(* IEC 61131-3 sources: POMIRTS_lab3/AS/Library/LoopCont/V3.03.2, 3 files *)

(* ---- LoopCont.typ ---- *)
(********************************************************************
 * COPYRIGHT (C) BERNECKER + RAINER, AUSTRIA, A-5142 EGGELSBERG
 ********************************************************************
 * Library: LoopCont
 * File: LoopCont.typ
 * Created: 11.11.2003
 ********************************************************************
 * Global data types of library LoopCont
 ********************************************************************)

TYPE
	lcslimpid_par_typ : 	STRUCT
		Y_max : INT;
		Y_min : INT;
		Kp : REAL;
		Tn : REAL;
		Tv : REAL;
		Kfbk : REAL;
	END_STRUCT;
	lcpid_tune_addpar_typ : 	STRUCT
		t_max_tune : UDINT;
		dY_max : REAL;
		Tf_Tv : REAL;
		Kw : REAL;
		Kfbk : REAL;
		fbk_mode : USINT;
		d_mode : USINT;
		calc_mode : USINT;
	END_STRUCT;
	lcpid_tune_osc_options_typ : 	STRUCT
		osc_minAmplitude : INT;
		Q_min : REAL;
	END_STRUCT;
	lcpid_osc_val_typ : 	STRUCT
		X : INT;
		t : UDINT;
	END_STRUCT;
	lcpid_osc_per_typ : 	STRUCT
		max : lcpid_osc_val_typ;
		min : lcpid_osc_val_typ;
	END_STRUCT;
	lcpid_tune_osc_typ : 	STRUCT
		options : lcpid_tune_osc_options_typ;
		oscPhase : UINT;
		dir : SINT;
		Y_hi : INT;
		Y_lo : INT;
		i_maxPeriod : UINT;
		i_period : UINT;
		X_ampl : DINT;
		X_avg : DINT;
		X_min_avg : DINT;
		X_max_avg : DINT;
		Y_avg : DINT;
		deltaY : DINT;
		t_Ylohi : ARRAY[0..4] OF UDINT;
		t_Yhilo : ARRAY[0..4] OF UDINT;
		Q_act : REAL;
		a_wx : INT;
		amplitudeRatio : REAL;
		Ku : REAL;
		tPeriod : UDINT;
		period : ARRAY[0..4] OF lcpid_osc_per_typ;
	END_STRUCT;
	lcpid_tune_step_options_typ : 	STRUCT
		eqDeltaX : INT;
		eqDeltaWX : INT;
		eqDeltat : UDINT;
		evalDeltaX : INT;
		evalNfilter : UINT;
		exitNotMaxdXCount : UINT;
		exitdXRatio : UINT;
	END_STRUCT;
	lcpid_tune_step_typ : 	STRUCT
		options : lcpid_tune_step_options_typ;
		Y0 : INT;
		Y1 : INT;
		t_jump : UDINT;
		W : INT;
		X0 : INT;
		Xmax : INT;
		Xmin : INT;
		Xfiltered : DINT;
		deltaXok : BOOL;
		deltaWXok : BOOL;
		eqTime : UDINT;
		dir : SINT;
		deltaX : INT;
		X1 : INT;
		t1 : UDINT;
		t1set : BOOL;
		dX_dt : REAL;
		dX_dt_max : REAL;
		XmaxGrad : INT;
		maxX1 : INT;
		maxX2 : INT;
		maxt1 : UDINT;
		maxt2 : UDINT;
		tmaxGrad : UDINT;
		gainFactor : REAL;
		deadTime : UDINT;
		riseTime : UDINT;
		notMaxCount : UINT;
		gradientRatio : UINT;
		cycleTime : UDINT;
	END_STRUCT;
	lcdblpid_tune_typ : 	STRUCT
		P1_manualAdjust : INT;
		I1_manualAdjust : INT;
		D1_manualAdjust : INT;
		P2_manualAdjust : INT;
		I2_manualAdjust : INT;
		D2_manualAdjust : INT;
		X_min : INT;
		X_max : INT;
		X0 : INT;
		de_min : INT;
		Y0 : INT;
		Y1step : INT;
		Y2step : INT;
		tuneY1_opt : UDINT;
		tuneY2_opt : UDINT;
		tune_first : USINT;
		hyst : INT;
		measDelta : INT;
		osc_opt : lcpid_tune_osc_options_typ;
		step_opt : lcpid_tune_step_options_typ;
	END_STRUCT;
	lcdblpid_par_typ : 	STRUCT
		Y_max : INT;
		Y_min : INT;
		K_fact : INT;
		Kp : REAL;
		Tn : REAL;
		Tv : REAL;
	END_STRUCT;
	lcCurveByPoints_TabEntry_type : 	STRUCT
		x : INT;
		y : INT;
	END_STRUCT;
	lcpid_addPar_typ : 	STRUCT
		y_autotune_on : INT;
		y_autotune_off : INT;
		t_autotune_max : UDINT;
		diff_dx_max : INT;
		diff_dt_max : UDINT;
		osc_nrPeriods : UINT;
		osc_minAmplitude : INT;
		optSwitches : UINT;
		dY_max : REAL;
		Tf_Tv : REAL;
		Kw : REAL;
		Kfbk : REAL;
		fbk_mode : USINT;
		d_mode : USINT;
		calc_mode : USINT;
	END_STRUCT;
	lcpid_internal_typ : 	STRUCT
		size : UINT;
		valid : BOOL;
		autotune_addpar : lcpid_addPar_typ;
		Y_max : INT;
		Y_min : INT;
		dY_max1 : DINT;
		Kp1 : DINT;
		Kp_Tn_1 : DINT;
		Tv_Tf_1 : DINT;
		Tf_reciproc_1 : DINT;
		Kw1 : DINT;
		Kfbk_Kp_1 : DINT;
		fbk_mode : USINT;
		d_mode : USINT;
		calc_mode : USINT;
		prescalerPow2 : UINT;
		force_outmode : USINT;
		Y_force : INT;
		W : INT;
		X : INT;
		pid_init : USINT;
		dt : UDINT;
		Yp1 : DINT;
		Yp2 : DINT;
		dYi1 : DINT;
		dYi2 : DINT;
		Yi1 : DINT;
		Yi2 : DINT;
		dt_Tf_1 : DINT;
		a11 : DINT;
		a12 : DINT;
		a21 : DINT;
		a22 : DINT;
		Yd1 : DINT;
		Yd2 : DINT;
		Ytotal1 : DINT;
		Ytotal2 : DINT;
		Ylim1 : DINT;
		Ylim2 : DINT;
		Y1 : DINT;
		Y2 : DINT;
		e_fbk : DINT;
	END_STRUCT;
	lcpid_osc_typ : 	STRUCT
		i_maxPeriod : UINT;
		i_period : UINT;
		X_amplitude : DINT;
		amplitudeRatio : REAL;
		tPeriod : UDINT;
		period : ARRAY[0..4] OF lcpid_osc_per_typ;
	END_STRUCT;
	lcpid_procPar_typ : 	STRUCT
		size : UINT;
		valid : BOOL;
		stepResp_valid : BOOL;
		stepResp_v : REAL;
		stepResp_t_u : UDINT;
		stepResp_t_g : UDINT;
		osc_valid : BOOL;
		osc_amplitudeRatio : REAL;
		osc_tPeriod : UDINT;
		force_params : BOOL;
		Kp : REAL;
		Kp_tune : REAL;
		Tn : REAL;
		Tn_tune : REAL;
		Tv : REAL;
		Tv_tune : REAL;
	END_STRUCT;
	lcpid_old_typ : 	STRUCT
		processPar : lcpid_procPar_typ;
		P_manualAdjust : INT;
		I_manualAdjust : INT;
		D_manualAdjust : INT;
		Y_min : INT;
		Y_max : INT;
		dY_max : REAL;
		Tf_Tv : REAL;
		Kw : REAL;
		Kfbk : REAL;
		request : UDINT;
		time : UDINT;
		W : INT;
		fbk_mode : USINT;
		d_mode : USINT;
		enable : BOOL;
	END_STRUCT;
	lcpid_stepResp_typ : 	STRUCT
		W_old : INT;
		dW : INT;
		x_prev : INT;
		x_inflectionPt : INT;
		t_inflectionPt : UDINT;
		v : REAL;
		v_max : REAL;
		t_u : UDINT;
		x_pre : INT;
		x_max : INT;
	END_STRUCT;
	lcpid_diff_typ : 	STRUCT
		init : BOOL;
		x_old : INT;
		dx : INT;
		dt : UDINT;
		dx_dt : REAL;
	END_STRUCT;
END_TYPE

(* ---- LoopCont.fun ---- *)
(********************************************************************
 * COPYRIGHT (C) BERNECKER + RAINER, AUSTRIA, A-5142 EGGELSBERG
 ********************************************************************
 * Library: LoopCont
 * File: LoopCont.fun
 * Created: 02.11.2006
 ********************************************************************
 * Functions and function blocks of library LoopCont
 ********************************************************************)

FUNCTION_BLOCK LCSlimPID (* PID controller with integrated tuning. *)
	VAR_INPUT
		enable : BOOL;
		W : INT;
		X : INT;
		request : UDINT;
		pPar : REFERENCE TO lcslimpid_par_typ;
		basetime : UDINT;
	END_VAR
	VAR_OUTPUT
		e : DINT;
		Y : INT;
		status : UINT;
		addInfo : UINT;
	END_VAR
	VAR
		MovAvgFlt_inst : LCMovAvFilter;
		PIDTune_inst : LCPIDTune;
		PID_inst : LCPID;
		enable_old : BOOL;
		requ_old : UDINT;
	END_VAR
END_FUNCTION_BLOCK

FUNCTION_BLOCK LCPWM (* Pulse width modulator. *)
	VAR_INPUT
		enable : BOOL;
		x : INT;
		max_value : INT;
		min_value : INT;
		t_min_pulse : UINT;
		t_period : UINT;
		basetime : UDINT;
	END_VAR
	VAR_OUTPUT
		status : UINT;
		pulse : BOOL;
	END_VAR
	VAR
		area : DINT;
		period : UINT;
		time_old : UDINT;
		last : UINT;
		x_old : INT;
		enable_old : BOOL;
	END_VAR
END_FUNCTION_BLOCK

FUNCTION_BLOCK LCContinServo (* Control of a continuous servo drive without position feedback. *)
	VAR_INPUT
		enable : BOOL;
		x : INT;
		max_value : INT;
		min_value : INT;
		t_impulse : UINT;
		t_change_up : UINT;
		t_change_down : UINT;
		ref : BOOL;
		basetime : UDINT;
	END_VAR
	VAR_OUTPUT
		status : UINT;
		up : BOOL;
		down : BOOL;
		hysteresis_up : UINT;
		hysteresis_down : UINT;
		refOk : BOOL;
	END_VAR
	VAR
		enable_old : BOOL;
		time_old : UDINT;
		ref_old : BOOL;
		t_cnt : DINT;
		y_fix31_1 : DINT;
		y_fix31_2 : DINT;
	END_VAR
END_FUNCTION_BLOCK

FUNCTION_BLOCK LCMinMax (* Smallest and largest peak value. *)
	VAR_INPUT
		reset : BOOL;
		in : INT;
	END_VAR
	VAR_OUTPUT
		out_min : INT;
		out_max : INT;
	END_VAR
END_FUNCTION_BLOCK

FUNCTION_BLOCK LCPIDTune (* Automatically determines the control parameters of an LCPID() instance with various methods and setting guidelines. *)
	VAR_INPUT
		enable : BOOL;
		Y_min : INT;
		Y_max : INT;
		Y0 : INT;
		Y1 : INT;
		okToStep : BOOL;
		X0 : INT;
		X_min : INT;
		X_max : INT;
		P_manualAdjust : INT;
		I_manualAdjust : INT;
		D_manualAdjust : INT;
		request : UDINT;
		basetime : UDINT;
		pAddPar : REFERENCE TO lcpid_tune_addpar_typ;
		pOptions_osc : REFERENCE TO lcpid_tune_osc_options_typ;
		pOptions_step : REFERENCE TO lcpid_tune_step_options_typ;
	END_VAR
	VAR_OUTPUT
		status : UINT;
		addInfo : UINT;
		ident : UDINT;
		state : UINT;
		rdyToStep : BOOL;
	END_VAR
	VAR
		dt : UDINT;
		t_autotune : UDINT;
		status_tmp : UINT;
		curveDown : BOOL;
		e : INT;
		e_minAmp : INT;
		e_old_up : INT;
		e_old_down : INT;
		curveUp : BOOL;
		e_old : INT;
		MovAvgFlt_inst : LCMovAvFilter;
		old : lcpid_old_typ;
		processPar : lcpid_procPar_typ;
		internal_data : lcpid_internal_typ;
		addPar : lcpid_tune_addpar_typ;
		oscillation : lcpid_tune_osc_typ;
		stepresponse : lcpid_tune_step_typ;
	END_VAR
END_FUNCTION_BLOCK

FUNCTION_BLOCK LCDblActPID (* PID controller with two outputs for two opposing manipulated variables and integrated tuning. *)
	VAR_INPUT
		enable : BOOL;
		W : INT;
		X : INT;
		Y_man : INT;
		hold_I : BOOL;
		mode : USINT;
		okToStep : BOOL;
		basetime : UDINT;
		pPar1 : REFERENCE TO lcdblpid_par_typ;
		pPar2 : REFERENCE TO lcdblpid_par_typ;
		pAddPar : REFERENCE TO lcpid_tune_addpar_typ;
		pOpt : REFERENCE TO lcdblpid_tune_typ;
	END_VAR
	VAR_OUTPUT
		e : DINT;
		Y1 : INT;
		Y2 : INT;
		status : UINT;
		tuneState : USINT;
		rdyToStep : BOOL;
	END_VAR
	VAR
		enable_old : BOOL;
		pid : LCPID;
		tune : LCPIDTune;
		gradient : REAL;
		Y_avg : DINT;
		tcnt : UDINT;
		Tmeas : INT;
		y_lim_old : INT;
		use_par : USINT;
		meas : USINT;
		mode_old : USINT;
		tune_step : USINT;
		tune_grad : USINT;
		tune_2nd : USINT;
		invert : USINT;
		mode_int : USINT;
	END_VAR
END_FUNCTION_BLOCK

FUNCTION_BLOCK LCPFM (* Pulse frequency modul. *)
	VAR_INPUT
		enable : BOOL;
		x : INT;
		max_value : INT;
		min_value : INT;
		t_pulse : UINT;
		t_pause : UINT;
		basetime : UDINT;
	END_VAR
	VAR_OUTPUT
		status : UINT;
		pulse : BOOL;
	END_VAR
	VAR
		enable_old : BOOL;
		range : INT;
		area : DINT;
		area_c : DINT;
		time_old : UDINT;
		last : DINT;
		tpls : DINT;
	END_VAR
END_FUNCTION_BLOCK

FUNCTION_BLOCK LCCurveByPoints (* y=f(x) function using coordinates. *)
	VAR_INPUT
		x : INT;
		NoOfPoints : UINT;
		ptr_table : REFERENCE TO lcCurveByPoints_TabEntry_type;
	END_VAR
	VAR_OUTPUT
		status : UINT;
		y : INT;
	END_VAR
	VAR
		i_tab : INT;
		iterations : UINT;
		scal1 : LCScINT;
	END_VAR
END_FUNCTION_BLOCK

FUNCTION_BLOCK LCPWM_DMod (* Pulse width modulator, see LCPWM(). *)
	VAR_INPUT
		enable : BOOL;
		x : INT;
		max_value : INT;
		min_value : INT;
		tminpuls : UINT;
		tperiod : UINT;
		basetime : UDINT;
	END_VAR
	VAR_OUTPUT
		status : UINT;
		y : BOOL;
	END_VAR
	VAR
		area : DINT;
		period : UINT;
		time_old : UDINT;
		last : UINT;
		x_old : INT;
		enable_old : BOOL;
	END_VAR
END_FUNCTION_BLOCK

FUNCTION_BLOCK LCPIDpara (* PID controller configuration. *)
	VAR_INPUT
		enable : BOOL;
		enter : BOOL;
		Y_max : INT;
		Y_min : INT;
		dY_max : REAL;
		Kp : REAL;
		Tn : REAL;
		Tv : REAL;
		Tf : REAL;
		Kw : REAL;
		Kfbk : REAL;
		fbk_mode : USINT;
		d_mode : USINT;
		calc_mode : USINT;
	END_VAR
	VAR_OUTPUT
		status : UINT;
		ident : UDINT;
	END_VAR
	VAR
		internal_data : lcpid_internal_typ;
	END_VAR
END_FUNCTION_BLOCK

FUNCTION_BLOCK LCRampLim (* Ramp generator with limitation. *)
	VAR_INPUT
		enable : BOOL;
		x : INT;
		tup : UINT;
		tdown : UINT;
		max_value : INT;
		min_value : INT;
		yset : INT;
		set : BOOL;
		basetime : UDINT;
	END_VAR
	VAR_OUTPUT
		status : UINT;
		y : INT;
		xreached : BOOL;
		max_limit : BOOL;
		min_limit : BOOL;
	END_VAR
	VAR
		time_old : UDINT;
		rest : UINT;
		enable_old : BOOL;
	END_VAR
END_FUNCTION_BLOCK

FUNCTION_BLOCK LCPID (* PID controller. *)
	VAR_INPUT
		enable : BOOL;
		ident : UDINT;
		W : INT;
		X : INT;
		A : INT;
		Y_man : INT;
		Y_fbk : INT;
		hold_I : BOOL;
		out_mode : USINT;
		basetime : UDINT;
	END_VAR
	VAR_OUTPUT
		status : UINT;
		e : DINT;
		Y : INT;
		Yp : DINT;
		Yi : DINT;
		Yd : DINT;
	END_VAR
	VAR
		time_old : UDINT;
		Tv_Tf_old : DINT;
		enable_old : BOOL;
		e_old : DINT;
	END_VAR
END_FUNCTION_BLOCK

FUNCTION_BLOCK LCTimeBasedOnOff (* 3-position step output, see LCContinServo(). *)
	VAR_INPUT
		enable : BOOL;
		x : INT;
		max_value : INT;
		min_value : INT;
		timpulse : UINT;
		tchange_up : UINT;
		tchange_dwn : UINT;
		ref : BOOL;
		basetime : UDINT;
	END_VAR
	VAR_OUTPUT
		status : UINT;
		up : BOOL;
		down : BOOL;
		hysteresis_up : UINT;
		hysteresis_dwn : UINT;
		refOK : BOOL;
	END_VAR
	VAR
		enable_old : BOOL;
		time_old : UDINT;
		ref_old : BOOL;
		t_cnt : DINT;
		y_fix31_1 : DINT;
		y_fix31_2 : DINT;
	END_VAR
END_FUNCTION_BLOCK

FUNCTION_BLOCK LCDifferentiate (* Differentiator with filter. *)
	VAR_INPUT
		enable : BOOL;
		x : INT;
		tv : UINT;
		tf : UINT;
		basetime : UDINT;
	END_VAR
	VAR_OUTPUT
		status : UINT;
		y : INT;
	END_VAR
	VAR
		time_old : UDINT;
		enable_old : BOOL;
		a2n : DINT;
		a1 : DINT;
	END_VAR
END_FUNCTION_BLOCK

FUNCTION_BLOCK LCPIDAutoTune (* Automatically determines the control parameters of an LCPID() instance with various methods and setting guidelines. *)
	VAR_INPUT
		enable : BOOL;
		Y_max : INT;
		Y_min : INT;
		P_manualAdjust : INT;
		I_manualAdjust : INT;
		D_manualAdjust : INT;
		request : USINT;
		basetime : UDINT;
	END_VAR
	VAR_OUTPUT
		status : UINT;
		ident : UDINT;
		addInfo : UINT;
		state : UINT;
	END_VAR
	VAR
		dt : UDINT;
		t_autotune : UDINT;
		diff : lcpid_diff_typ;
		old : lcpid_old_typ;
		stepResponse : lcpid_stepResp_typ;
		oscillation : lcpid_osc_typ;
		processPar : lcpid_procPar_typ;
		internal_data : lcpid_internal_typ;
	END_VAR
END_FUNCTION_BLOCK

FUNCTION_BLOCK LC2PHy (* 2-position element with hysteresis. *)
	VAR_INPUT
		enable : BOOL;
		x : INT;
		xstart : INT;
		xsetvalue : INT;
		hysteresis : UINT;
		ymax : INT;
		ymin : INT;
	END_VAR
	VAR_OUTPUT
		status : UINT;
		y : INT;
		y1 : BOOL;
	END_VAR
	VAR
		enable_old : BOOL;
		x_old : INT;
	END_VAR
END_FUNCTION_BLOCK

FUNCTION_BLOCK LCScUINT (* Scaling and limiting of unsigned integer signals. *)
	VAR_INPUT
		x : UINT;
		x1 : UINT;
		y1 : UINT;
		x2 : UINT;
		y2 : UINT;
	END_VAR
	VAR_OUTPUT
		y : UINT;
	END_VAR
END_FUNCTION_BLOCK

FUNCTION_BLOCK LC3PHy (* 3-position element with hysteresis. *)
	VAR_INPUT
		enable : BOOL;
		x : INT;
		xstart : INT;
		xsetvalue1 : INT;
		xsetvalue2 : INT;
		hysteresis1 : UINT;
		hysteresis2 : UINT;
		ymax : INT;
		ymid : INT;
		ymin : INT;
	END_VAR
	VAR_OUTPUT
		status : UINT;
		y : INT;
		ymx : BOOL;
		ymn : BOOL;
	END_VAR
	VAR
		enable_old : BOOL;
		x_old : INT;
	END_VAR
END_FUNCTION_BLOCK

FUNCTION_BLOCK LCComparator (* Comparator. *)
	VAR_INPUT
		enable : BOOL;
		xp : INT;
		xn : INT;
		sd : UINT;
	END_VAR
	VAR_OUTPUT
		greater : BOOL;
		equal : BOOL;
		lower : BOOL;
	END_VAR
END_FUNCTION_BLOCK

FUNCTION_BLOCK LCCounter (* Counting module for base time generation. *)
	VAR_OUTPUT
		muscnt : UDINT;
		mus100cnt : UDINT;
		mscnt : UDINT;
		ms100cnt : UDINT;
		seccnt : UDINT;
	END_VAR
	VAR
		state : UINT;
		sysinf_inst : SysInfo;
		musecs_old : UINT;
		bootkey_old : UDINT;
		sys_ticks_old : UDINT;
		to_100us : UDINT;
		to_1ms : UDINT;
		to_100ms : UINT;
		to_1s : UINT;
	END_VAR
END_FUNCTION_BLOCK

FUNCTION_BLOCK LCIntegrate (* Integrator with limits and set value. *)
	VAR_INPUT
		enable : BOOL;
		x : INT;
		tn : UINT;
		max_value : INT;
		min_value : INT;
		yset : INT;
		set : BOOL;
		basetime : UDINT;
	END_VAR
	VAR_OUTPUT
		status : UINT;
		y : INT;
		max_limit : BOOL;
		min_limit : BOOL;
	END_VAR
	VAR
		time_old : UDINT;
		rest : DINT;
		enable_old : BOOL;
	END_VAR
END_FUNCTION_BLOCK

FUNCTION_BLOCK LCLimit (* Limiter with overrun indicators. *)
	VAR_INPUT
		enable : BOOL;
		in : DINT;
		max_value : INT;
		min_value : INT;
	END_VAR
	VAR_OUTPUT
		status : UINT;
		out : INT;
		max_limit : BOOL;
		min_limit : BOOL;
	END_VAR
END_FUNCTION_BLOCK

FUNCTION_BLOCK LCLiScDINT (* Scaling and limiting of double integer signals. *)
	VAR_INPUT
		x : DINT;
		x1 : DINT;
		y1 : DINT;
		x2 : DINT;
		y2 : DINT;
	END_VAR
	VAR_OUTPUT
		y : DINT;
	END_VAR
END_FUNCTION_BLOCK

FUNCTION_BLOCK LCLiScINT (* Scaling and limiting of integer signals. *)
	VAR_INPUT
		x : INT;
		x1 : INT;
		y1 : INT;
		x2 : INT;
		y2 : INT;
	END_VAR
	VAR_OUTPUT
		y : INT;
	END_VAR
END_FUNCTION_BLOCK

FUNCTION_BLOCK LCLiScUINT (* Scaling and limiting of unsigned integer signals. *)
	VAR_INPUT
		x : UINT;
		x1 : UINT;
		y1 : UINT;
		x2 : UINT;
		y2 : UINT;
	END_VAR
	VAR_OUTPUT
		y : UINT;
	END_VAR
END_FUNCTION_BLOCK

FUNCTION_BLOCK LCMovAvFilter (* Floating average value filter. *)
	VAR_INPUT
		enable : BOOL;
		x : INT;
		base : UINT;
	END_VAR
	VAR_OUTPUT
		status : UINT;
		y : INT;
	END_VAR
	VAR
		sum_old : DINT;
		x_old_ptr : UDINT;
		x_old : ARRAY[0..31] OF INT;
		xIdx : UINT;
		base_old : UINT;
		enable_old : BOOL;
		bootkey_old : UDINT;
	END_VAR
END_FUNCTION_BLOCK

FUNCTION_BLOCK LCNegDINT (* Negation of double integer signals *)
	VAR_INPUT
		in : DINT;
	END_VAR
	VAR_OUTPUT
		out : DINT;
	END_VAR
END_FUNCTION_BLOCK

FUNCTION_BLOCK LCNegINT (* Negation of integer signals. *)
	VAR_INPUT
		in : INT;
	END_VAR
	VAR_OUTPUT
		out : INT;
	END_VAR
END_FUNCTION_BLOCK

FUNCTION_BLOCK LCNegPeakVal (* Negative peak value, see LCMinMax(). *)
	VAR_INPUT
		in : INT;
		reset : BOOL;
	END_VAR
	VAR_OUTPUT
		out : INT;
	END_VAR
END_FUNCTION_BLOCK

FUNCTION_BLOCK LCPosPeakVal (* Positive peak value, see LCMinMax(). *)
	VAR_INPUT
		in : INT;
		reset : BOOL;
	END_VAR
	VAR_OUTPUT
		out : INT;
	END_VAR
END_FUNCTION_BLOCK

FUNCTION_BLOCK LCPT1 (* First-order delay element. *)
	VAR_INPUT
		enable : BOOL;
		x : INT;
		t : UINT;
		yset : INT;
		set : BOOL;
		basetime : UDINT;
	END_VAR
	VAR_OUTPUT
		status : UINT;
		y : INT;
	END_VAR
	VAR
		time_old : UDINT;
		rest : DINT;
		enable_old : BOOL;
	END_VAR
END_FUNCTION_BLOCK

FUNCTION_BLOCK LCScDINT (* Scaling of double integer signals. *)
	VAR_INPUT
		x : DINT;
		x1 : DINT;
		y1 : DINT;
		x2 : DINT;
		y2 : DINT;
	END_VAR
	VAR_OUTPUT
		y : DINT;
	END_VAR
END_FUNCTION_BLOCK

FUNCTION_BLOCK LCScINT (* Scaling of integer signals. *)
	VAR_INPUT
		x : INT;
		x1 : INT;
		y1 : INT;
		x2 : INT;
		y2 : INT;
	END_VAR
	VAR_OUTPUT
		y : INT;
	END_VAR
END_FUNCTION_BLOCK

(* ---- LoopCont.var ---- *)
(********************************************************************
 * COPYRIGHT (C) BERNECKER + RAINER, AUSTRIA, A-5142 EGGELSBERG
 ********************************************************************
 * Library: LoopCont
 * File: LoopCont.var
 * Created: 02.11.2006
 ********************************************************************
 * Constants of library LoopCont
 ********************************************************************)
VAR CONSTANT
	LC_ERR_LCPIDTune_INVALID_REQUEST : UINT := 31559;
	LCPIDAUTOTUNE_STATE_STEPRESPONSE : UINT := 20;
	LCPIDAUTOTUNE_ADDINFO_OSC_PERIOD : UINT := 101;
	LCPIDAUTOTUNE_STATE_RESET_CTRLR : UINT := 49;
	LCPIDAUTOTUNE_REQU_STEPRESPONSE : USINT := 1;
	LCPIDAUTOTUNE_OPT_NEW_WEIGHTING : UINT := 4;
	LCPIDAUTOTUNE_ADDINFO_PRESCALER : UINT := 102;
	LC_ERR_LCPIDAutotune_W_CHANGED : UINT := 12041;
	LC_ERR_LCPIDAutotune_PARAMETER : UINT := 12039;
	LCPID_TUNE_STATE_OSC_WAIT_NEXT : UINT := 14;
	LCPID_TUNE_STATE_OSC_PERFORM_2 : UINT := 13;
	LCPID_TUNE_STATE_OSC_PERFORM_1 : UINT := 12;
	LCPID_OUT_MODE_FREEZE_JOLTFREE : USINT := 105;
	LCPIDAUTOTUNE_ADDINFO_OSC_AMPL : UINT := 100;
	LC_ERR_LCTimBasOnOff_TIMPULSE : UINT := 12036;
	LC_ERR_LCContinServo_TIMPULSE : UINT := 12036;
	LCPID_TUNE_STATE_STEP_WAITEQ2 : UINT := 22;
	LCPID_TUNE_STATE_STEP_WAITEQ1 : UINT := 20;
	LCPID_TUNE_STATE_STEP_MAXGRAD : UINT := 21;
	LCPID_TUNE_STATE_OSC_SEQ_CNTL : UINT := 11;
	LCPID_TUNE_ADDINFO_OSC_PERIOD : UINT := 111;
	LCPID_OUT_MODE_CLOSE_JOLTFREE : USINT := 104;
	LCPIDAUTOTUNE_STATE_WAIT_STEP : UINT := 10;
	LCPIDAUTOTUNE_STATE_OSCILLATE : UINT := 40;
	LC_WARN_LCDBLPID_TUNE_CHANGE : UINT := 12019;
	LC_ERR_LCTimBasOnOff_TCHANGE : UINT := 12035;
	LC_ERR_LCPIDTune_CONTROL_VAR : UINT := 31560;
	LC_ERR_LCPIDAutotune_TIMEOUT : UINT := 12040;
	LC_ERR_LCCurveByPoints_TABLE : UINT := 12045;
	LC_ERR_LCContinServo_TCHANGE : UINT := 12035;
	LCPID_TUNE_STATE_OSC_CNTLPAR : UINT := 19;
	LCPID_TUNE_REQU_STEPRESPONSE : UDINT := 2;
	LCPID_TUNE_ADDINFO_PRESCALER : UINT := 112;
	LCPID_OUT_MODE_OPEN_JOLTFREE : USINT := 103;
	LCPIDAUTOTUNE_STATE_WAIT_MAX : UINT := 30;
	LCPIDAUTOTUNE_STATE_FINISHED : UINT := 50;
	LCPIDAUTOTUNE_REQU_OSCILLATE : USINT := 2;
	LC_WARN_LCPIDTune_CYCLETIME : UINT := 12004;
	LCSLIMPID_REQU_STEPRESPONSE : UDINT := 2;
	LCPID_TUNE_STATE_RESET_CNTL : UINT := 49;
	LCPID_TUNE_REQU_CHR_DIST_OS : UDINT := 2000;
	LCPID_TUNE_REQU_CHR_DIST_AP : UDINT := 1000;
	LCPID_OUT_MODE_MAN_JOLTFREE : USINT := 102;
	LCPID_FBK_MODE_EXT_SELECTOR : USINT := 3;
	LCPIDAUTOTUNE_REQU_AUTOTUNE : USINT := 3;
	LCPIDAUTOTUNE_ADDINFO_Y_OFF : UINT := 103;
	LC_ERR_LCRampLim_TUP_TDOWN : UINT := 12034;
	LC_ERR_LCPWM_DMod_TMINPULS : UINT := 12032;
	LC_ERR_LCPID_PAR_PRESCALER : UINT := 12042;
	LC_ERR_LCPIDTune_W_CHANGED : UINT := 12041;
	LC_ERR_LCPIDTune_PARAMETER : UINT := 12039;
	LC_ERR_LCPIDAutotune_ABORT : UINT := 12038;
	LCSLIMPID_REQU_WRITE_PARAS : UDINT := 4;
	LCSLIMPID_REQU_CHR_DIST_OS : UDINT := 2000;
	LCSLIMPID_REQU_CHR_DIST_AP : UDINT := 1000;
	LCPID_TUNE_STATE_OSCILLATE : UINT := 10;
	LCPID_TUNE_STATE_CALC_PARA : UINT := 45;
	LCPID_TUNE_REQU_CHR_REF_OS : UDINT := 5000;
	LCPID_TUNE_REQU_CHR_REF_AP : UDINT := 4000;
	LCPIDAUTOTUNE_ADDINFO_Y_ON : UINT := 104;
	LC_ERR_LCPWM_DMod_TPERIOD : UINT := 12033;
	LC_ERR_LCPID_PAR_CALCMODE : UINT := 31555;
	LC_ERR_LCPIDTune_BASETIME : UINT := 31566;
	LC_ERR_LCMovAvFilter_BASE : UINT := 31551;
	LCSLIMPID_REQU_READ_PARAS : UDINT := 3;
	LCSLIMPID_REQU_CHR_REF_OS : UDINT := 5000;
	LCSLIMPID_REQU_CHR_REF_AP : UDINT := 4000;
	LCPID_TUNE_STATE_FINISHED : UINT := 50;
	LCPID_TUNE_REQU_OSCILLATE : UDINT := 1;
	LCPIDAUTOTUNE_STATE_READY : UINT := 0;
	LC_WARN_LCPID_YFBK_LIMIT : UINT := 12003;
	LC_WARN_LCPID_I_MINLIMIT : UINT := 12002;
	LC_WARN_LCPID_I_MAXLIMIT : UINT := 12001;
	LC_ERR_LCPID_PAR_FBKMODE : UINT := 31558;
	LC_ERR_LCPIDTune_TIMEOUT : UINT := 12040;
	LCSLIMPID_REQU_OSCILLATE : UDINT := 1;
	LCDBLPID_TSTATE_FINISHED : USINT := 3;
	LC_ERR_LCPIDTune_MAXMIN : UINT := 31564;
	LC_ERR_LC3PHy_XSETVALUE : UINT := 31565;
	LCPID_TUNE_REQU_ZN_DIST : UDINT := 3000;
	LCPID_TUNE_REQU_DIR_POS : UDINT := 10;
	LCPID_TUNE_REQU_DIR_NEG : UDINT := 20;
	LC_ERR_LCPID_PAR_DYMAX : UINT := 31557;
	LC_ERR_LCPID_PAR_DMODE : UINT := 31556;
	LC_ERR_LCPIDTune_ABORT : UINT := 12038;
	LC_ERR_LCDBLPID_WX_LOW : UINT := 31561;
	LCSLIMPID_REQU_ZN_DIST : UDINT := 3000;
	LCSLIMPID_REQU_DIR_POS : UDINT := 10;
	LCSLIMPID_REQU_DIR_NEG : UDINT := 20;
	LCPID_TUNE_STATE_READY : UINT := 0;
	LCPIDAUTOTUNE_REQU_OFF : USINT := 0;
	LC_WARN_LCxPHy_XSTART : UINT := 12006;
	LC_ERR_LCPWM_TMINPULS : UINT := 12032;
	LC_ERR_LCPID_PAR_KFBK : UINT := 12025;
	LC_ERR_LCIntegrate_TN : UINT := 31550;
	LC_ERR_LCDBLPID_DX_DT : UINT := 31562;
	LCPID_TUNE_REQU_PER_5 : UDINT := 500000;
	LCPID_TUNE_REQU_PER_4 : UDINT := 400000;
	LCPID_TUNE_REQU_PER_3 : UDINT := 300000;
	LCPID_TUNE_REQU_OSC_3 : UDINT := 30000;
	LCPID_TUNE_REQU_OSC_2 : UDINT := 20000;
	LCPID_TUNE_REQU_OSC_1 : UDINT := 10000;
	LCPID_OUT_MODE_FREEZE : USINT := 5;
	LCPID_FBK_MODE_INTERN : USINT := 1;
	LCPID_FBK_MODE_EXTERN : USINT := 2;
	LCPID_CALC_MODE_EXACT : USINT := 1;
	LCDBLPID_TSTATE_ERROR : USINT := 4;
	LCDBLPID_MODE_TUNE_Y2 : USINT := 9;
	LCDBLPID_MODE_TUNE_Y1 : USINT := 8;
	LC_ERR_LCPWM_TPERIOD : UINT := 12033;
	LC_ERR_LCPID_PARADAT : UINT := 31554;
	LC_ERR_LCPID_OUTMODE : UINT := 31553;
	LCSLIMPID_REQU_PER_5 : UDINT := 500000;
	LCSLIMPID_REQU_PER_4 : UDINT := 400000;
	LCSLIMPID_REQU_PER_3 : UDINT := 300000;
	LCSLIMPID_REQU_OSC_3 : UDINT := 30000;
	LCSLIMPID_REQU_OSC_2 : UDINT := 20000;
	LCSLIMPID_REQU_OSC_1 : UDINT := 10000;
	LCPID_OUT_MODE_CLOSE : USINT := 4;
	LCPID_CALC_MODE_FAST : USINT := 2;
	LCDBLPID_MODE_TUNE_6 : USINT := 7;
	LCDBLPID_MODE_TUNE_4 : USINT := 6;
	LC_WARN_DT_MAXLIMIT : UINT := 12000;
	LC_ERR_LCPID_PAR_TV : UINT := 12030;
	LC_ERR_LCPID_PAR_TN : UINT := 12029;
	LC_ERR_LCPID_PAR_TF : UINT := 12028;
	LC_ERR_LCPID_PAR_KW : UINT := 12027;
	LC_ERR_LCPID_PAR_KP : UINT := 12026;
	LCPID_TUNE_REQU_PID : UDINT := 100;
	LCPID_TUNE_REQU_OFF : UDINT := 0;
	LCPID_OUT_MODE_OPEN : USINT := 3;
	LCPID_OUT_MODE_AUTO : USINT := 1;
	LCDBLPID_TSTATE_OFF : USINT := 0;
	LC_ERR_LCPID_IDENT : UINT := 31552;
	LCSLIMPID_REQU_PID : UDINT := 100;
	LCSLIMPID_REQU_OFF : UDINT := 0;
	LCPID_TUNE_REQU_PI : UDINT := 200;
	LCPID_OUT_MODE_OFF : USINT := 0;
	LCPID_OUT_MODE_MAN : USINT := 2;
	LCDBLPID_TSTATE_Y2 : USINT := 2;
	LCDBLPID_TSTATE_Y1 : USINT := 1;
	LCSLIMPID_REQU_PI : UDINT := 200;
	LCPID_TUNE_REQU_P : UDINT := 300;
	LCSLIMPID_REQU_P : UDINT := 300;
	LC_ERR_DISABLED : UINT := 65534;
	LC_ERR_POINTER : UINT := 31563;
	LC_ERR_LCPT1_T : UINT := 12031;
	LCPID_D_MODE_X : USINT := 1;
	LCPID_D_MODE_E : USINT := 2;
	LC_WARN_Tx_DT : UINT := 12007;
	LC_ERR_MAXMIN : UINT := 12037;
	LC_ERROR : UINT := 12025;
END_VAR
